Fanuc TP program (LS listing): TEST.LS

/PROG  TEST
/ATTR
OWNER		= MNEDITOR;
COMMENT		= "";
PROG_SIZE	= 281;
CREATE		= DATE 21-09-08  TIME 22:35:38;
MODIFIED	= DATE 21-10-08  TIME 06:39:56;
FILE_NAME	= ;
VERSION		= 0;
LINE_COUNT	= 7;
MEMORY_SIZE	= 641;
PROTECT		= READ_WRITE;
TCD:  STACK_SIZE	= 0,
      TASK_PRIORITY	= 50,
      TIME_SLICE	= 0,
      BUSY_LAMP_OFF	= 0,
      ABORT_REQUEST	= 0,
      PAUSE_REQUEST	= 0;
DEFAULT_GROUP	= 1,*,*,*,*;
CONTROL_CODE	= 00000000 00000000;
/APPL

AUTO_SINGULARITY_HEADER;
  ENABLE_SINGULARITY_AVOIDANCE   : TRUE;
/MN
   1:L PR[8] 100mm/sec FINE Tool_Offset,PR[84]    ;
   2:   ;
   3:  SOFTFLOAT[1] ;
   4:L PR[6:INT_OnPart_HD1] 100mm/sec FINE Tool_Offset,PR[84]    ;
   5:  CALL HD1_CLOSE    ;
   6:  CALL GRIP_OPEN    ;
   7:  SOFTFLOAT END ;
/POS
/END
